FUNCTION_BLOCK fb_gm_transport
VAR_INPUT
END_VAR
VAR_OUTPUT
END_VAR
VAR
	SFCInit : bool;
	trn_lensPickUpDone: BOOL;
	trn_transportDone: BOOL;
	trn_lensSetDone: BOOL;
	var_process: INT;
	trn_homeDone: BOOL;
	trn_closeCheckDone: BOOL;
	trn_waittingLensDone: BOOL;
	retryTimer: TON;
	var_retryTimes: INT;
END_VAR

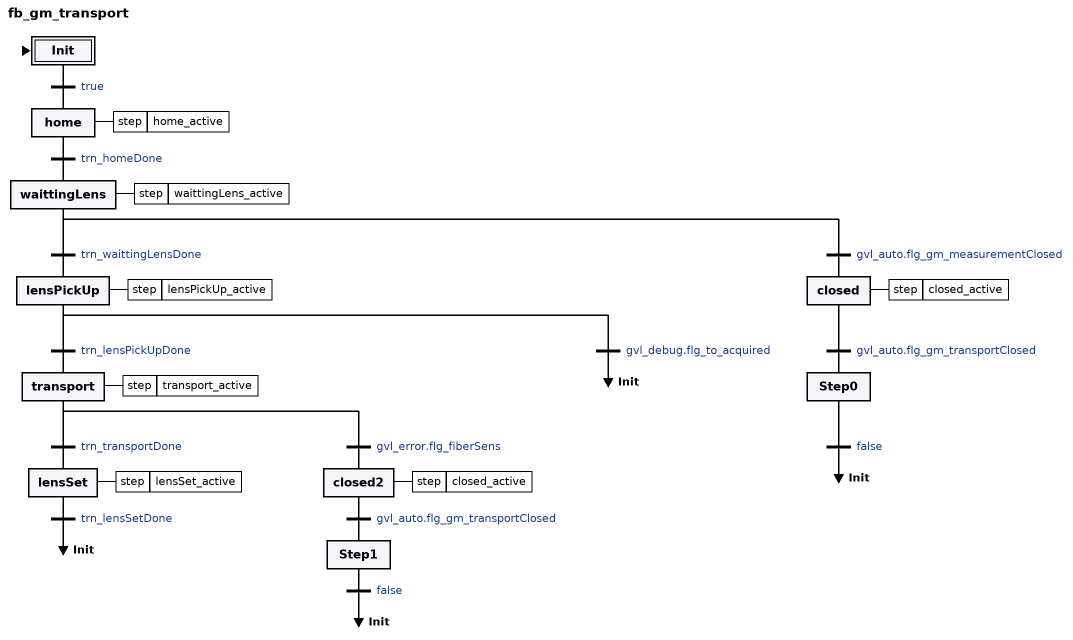
INITIAL_STEP Init:
END_STEP
TRANSITION FROM Init TO home
    := true;
END_TRANSITION
STEP home:
    home_active(N);  // step action
END_STEP
TRANSITION FROM home TO waittingLens
    := trn_homeDone;
END_TRANSITION
STEP waittingLens:
    waittingLens_active(N);  // step action
END_STEP
TRANSITION FROM waittingLens TO lensPickUp
    := trn_waittingLensDone;
END_TRANSITION
STEP lensPickUp:
    lensPickUp_active(N);  // step action
END_STEP
TRANSITION FROM lensPickUp TO transport
    := trn_lensPickUpDone;
END_TRANSITION
TRANSITION FROM lensPickUp TO Init
    := gvl_debug.flg_to_acquired;
END_TRANSITION
TRANSITION FROM waittingLens TO closed
    := gvl_auto.flg_gm_measurementClosed;
END_TRANSITION
STEP closed:
    closed_active(N);  // step action
END_STEP
TRANSITION FROM closed TO Step0
    := gvl_auto.flg_gm_transportClosed;
END_TRANSITION
STEP Step0:
END_STEP
TRANSITION FROM Step0 TO Init
    := false;
END_TRANSITION
STEP transport:
    transport_active(N);  // step action
END_STEP
TRANSITION FROM transport TO lensSet
    := trn_transportDone;
END_TRANSITION
STEP lensSet:
    lensSet_active(N);  // step action
END_STEP
TRANSITION FROM lensSet TO Init
    := trn_lensSetDone;
END_TRANSITION
TRANSITION FROM transport TO closed2
    := gvl_error.flg_fiberSens;
END_TRANSITION
STEP closed2:
    closed_active(N);  // step action
END_STEP
TRANSITION FROM closed2 TO Step1
    := gvl_auto.flg_gm_transportClosed;
END_TRANSITION
STEP Step1:
END_STEP
TRANSITION FROM Step1 TO Init
    := false;
END_TRANSITION

ACTION closed_active:
IF closed._x AND closed.x = FALSE THEN
	gvl_auto.flg_gm_transportClosed := FALSE;
ELSIF closed._x AND closed.x THEN
	gvl_auto.flg_gm_transportClosed := TRUE;
END_IF
END_ACTION

ACTION home_active:
IF home._x AND home.x = FALSE THEN
	var_process := 0;
	trn_homeDone := FALSE;
	gvl_debug.flg_to_demand:= FALSE;
ELSIF home._x AND home.x THEN
	CASE var_process OF 
		0:
			gvl_elecylinder.fbi_gm_axisPickUp.in_flg_run := FALSE;
			gvl_elecylinder.fbi_gm_axisPickUp.in_var_moveMode := eP_eleMoveMode.eleA;
			gvl_elecylinder.fbi_gm_axisTransport.in_flg_run := FALSE;
			gvl_elecylinder.fbi_gm_axisTransport.in_var_moveMode := eP_eleMoveMode.eleA;
			gvl_axis.ref_r.Execute := FALSE;
			gvl_axis.ref_r.Position := gvl_param.var_productInfo[gvl_param.var_currentProductID].teachPos.gm_rotary.origin;
			var_process := 1;
		1:
			gvl_elecylinder.fbi_gm_axisPickUp.in_flg_run := TRUE;
			gvl_elecylinder.fbi_gm_axisTransport.in_flg_run := TRUE;
			var_process := 2;
		2:
			IF gvl_elecylinder.ref_gm_axisPickUp.input.in_flg_sensA AND gvl_elecylinder.ref_gm_axisTransport.input.in_flg_sensA THEN
				gvl_elecylinder.fbi_gm_axisPickUp.in_flg_run := FALSE;
				gvl_elecylinder.fbi_gm_axisTransport.in_flg_run := FALSE;
				var_process := 3;
			END_IF
		3:
			gvl_solv.fbi_gm_pickup.in_flg_run := FALSE;
			gvl_solv.fbi_gm_pickup.in_var_moveMode := eP_svMoveMode.svA;
			var_process := 4;
		4:
			gvl_solv.fbi_gm_pickup.in_flg_run := TRUE;
			IF gvl_solv.ref_gm_pickUp.in.in_flg_sensA  THEN
				var_process := 5;
			END_IF
		5:
			gvl_auto.flg_gm_eleIsDown := FALSE;
			gvl_axis.ref_r.Execute := TRUE;
			IF gvl_axis.ref_r.Done THEN
				gvl_axis.ref_r.Execute := FALSE;
				var_process :=6;
			END_IF
		6:
			gvl_solv.fbi_gm_rotary.in_flg_run := FALSE;
			gvl_solv.fbi_gm_rotary.in_var_moveMode := eP_svMoveMode.svA;
			var_process := 7;
		7:
			gvl_solv.fbi_gm_rotary.in_flg_run := TRUE;
			IF gvl_solv.ref_gm_rotary.in.in_flg_sensA THEN
				var_process := 8;
			END_IF
		8:	
				trn_homeDone := TRUE;			
	END_CASE
END_IF
END_ACTION

ACTION lensPickUp_active:
IF lensPickUp._x AND lensPickUp.x = FALSE THEN
	gvl_axis.ref_r.Execute := FALSE;
	retryTimer.IN := FALSE;
	var_process := 0;
	var_retryTimes := 0;
	trn_lensPickUpDone := FALSE;
	gvl_auto.flg_gm_VacuumRetry := FALSE;
	gvl_solv.fbi_gm_ejector.in_flg_run := FALSE;
	gvl_solv.fbi_gm_pickup.in_flg_run := FALSE;
	gvl_solv.fbi_gm_rotary.in_flg_run := FALSE;
	gvl_elecylinder.fbi_gm_axisPickUp.in_flg_run := FALSE;
	gvl_axis.ref_r.Execute := FALSE;
ELSIF lensPickUp._x AND lensPickUp.x THEN
	CASE var_process OF 
		0:
			gvl_axis.ref_r.Position := gvl_param.var_productInfo[gvl_param.var_currentProductID].teachPos.gm_rotary.pickUp;
			gvl_axis.ref_r.Execute := TRUE;
			gvl_solv.fbi_gm_ejector.in_var_vacMode := eP_ejeVacMode.vacON;
			gvl_solv.fbi_gm_ejector.in_flg_run := TRUE;
			var_process := 1;
		1://axis theta move to pick up position
			gvl_solv.fbi_gm_ejector.in_flg_run := FALSE;
			IF gvl_axis.ref_r.Done THEN
				gvl_axis.ref_r.Execute := FALSE;
				var_process := 2;
			END_IF
		2:
			IF gvl_solv.ref_gm_ejctor.input.in_flg_sensVac THEN
				var_process := 3;
			END_IF
		3:
			gvl_solv.fbi_gm_chuck.in_var_moveMode := eP_svMoveMode.svA;
			gvl_solv.fbi_gm_push.in_var_moveMode := eP_svMoveMode.svA;
			gvl_solv.fbi_gm_chuck.in_flg_run := TRUE;
			gvl_solv.fbi_gm_push.in_flg_run := TRUE;
			var_process := 4;
		4:
			IF gvl_solv.ref_gm_chuck.in.in_flg_sensA AND gvl_solv.ref_gm_push.in.in_flg_sensA THEN
				gvl_solv.fbi_gm_chuck.in_flg_run := FALSE;
				gvl_solv.fbi_gm_push.in_flg_run := FALSE;
				var_process := 5;
			END_IF
		5:
			gvl_solv.fbi_gm_pickup.in_var_moveMode := eP_svMoveMode.svB;
			gvl_solv.fbi_gm_pickup.in_flg_run := TRUE;
			var_process := 6;
		6:
			IF gvl_solv.fbi_gm_pickup.out_flg_Done THEN
				gvl_solv.fbi_gm_pickup.in_flg_run := FALSE;
				var_process := 7;
			END_IF
		7:
			gvl_axis.ref_r.Position := gvl_param.var_productInfo[gvl_param.var_currentProductID].teachPos.gm_rotary.set;
			gvl_axis.ref_r.Execute := TRUE;
			var_process := 8;
		8:
			IF gvl_axis.ref_r.Done THEN
				gvl_axis.ref_r.Execute := FALSE;
				var_process := 9;	
			END_IF
		9:
			gvl_solv.fbi_gm_pickup.in_var_moveMode := eP_svMoveMode.svA;
			gvl_solv.fbi_gm_pickup.in_flg_run := TRUE;
			var_process := 10;
		10:
			IF gvl_solv.fbi_gm_pickup.out_flg_Done THEN
				gvl_solv.fbi_gm_pickup.in_flg_run := FALSE;
				var_process := 11;
			END_IF
		11:
			gvl_solv.fbi_gm_rotary.in_flg_run := FALSE;
			gvl_solv.fbi_gm_rotary.in_var_moveMode := eP_svMoveMode.svB;
			var_process:= 12;
		12:
			gvl_solv.fbi_gm_rotary.in_flg_run := TRUE;
			var_process := 13;
		13:
			IF gvl_solv.fbi_gm_rotary.out_flg_Done THEN
				gvl_solv.fbi_gm_rotary.in_flg_run := FALSE;
				var_process := 14;
			END_IF
		14:
			gvl_solv.fbi_gm_pickup.in_var_moveMode := eP_svMoveMode.svB;
			gvl_solv.fbi_gm_pickup.in_flg_run := TRUE;
			var_process := 15;
		15:
			IF gvl_solv.fbi_gm_pickup.out_flg_Done THEN
				gvl_solv.fbi_gm_pickup.in_flg_run := FALSE;
				var_process := 16;
			END_IF
		16:
			gvl_gm.flg_lensPickUpDone := TRUE;
			gvl_gm.var_buf_tranportCav := gvl_gm.var_buf_measurementCav;
			gvl_gm.flg_buf_gateLengthIsPassed := gvl_gm.flg_gateLengthIsPassed;
			var_process := 17;
		17:
			IF gvl_gm.flg_lensRequest AND NOT gvl_auto.flg_axisIsPcikingUp THEN
				IF gvl_debug.flg_check_quality AND gvl_debug.flg_to_stocker THEN
					gvl_debug.flg_to_demand:= TRUE;
				ELSE
					trn_lensPickUpDone := TRUE;		
				END_IF
			END_IF		
	END_CASE
END_IF
END_ACTION

ACTION lensSet_active:
IF lensSet._x AND lensSet.x = FALSE THEN
	trn_lensSetDone := FALSE;
	var_process := 0;
ELSIF lensSet._x AND lensSet.x THEN
	CASE var_process OF
		0:
			gvl_solv.fbi_gm_ejector.in_var_vacMode := eP_ejeVacMode.break;
			gvl_solv.fbi_gm_ejector.in_flg_run := FALSE;
			gvl_elecylinder.fbi_gm_axisPickUp.in_var_moveMode := eP_eleMoveMode.eleA;
			gvl_elecylinder.fbi_gm_axisPickUp.in_flg_run := FALSE;
			var_process := 1;
		1:
			gvl_solv.fbi_gm_ejector.in_flg_run := TRUE;
			IF gvl_solv.fbi_gm_ejector.out_flg_Done THEN
				gvl_solv.fbi_gm_ejector.in_flg_run := FALSE;
				var_process := 2;
			END_IF
		2:
			gvl_elecylinder.fbi_gm_axisPickUp.in_flg_run := TRUE;
			IF gvl_elecylinder.fbi_gm_axisPickUp.out_flg_Done THEN
				gvl_elecylinder.fbi_gm_axisPickUp.in_flg_run := FALSE;
				var_process := 3;
			END_IF
		3:
			gvl_gm.flg_lensSetDoneFromGM := TRUE;
			trn_lensSetDone := TRUE;
	END_CASE
END_IF
END_ACTION

PROPERTY p_Init : bool
GET
p_init := THIS^.SFCInit;
END_GET
SET
THIS^.SFCInit := p_init;
END_SET
END_PROPERTY

ACTION transport_active:
IF transport._x AND transport.x = FALSE THEN
	var_process := 0;
	trn_transportDone := FALSE;
	gvl_elecylinder.fbi_gm_axisTransport.in_flg_run := FALSE;
	gvl_elecylinder.fbi_gm_axisTransport.in_var_moveMode := eP_eleMoveMode.eleB;
	gvl_elecylinder.fbi_gm_axisPickUp.in_flg_run := FALSE;
	gvl_elecylinder.fbi_gm_axisPickUp.in_var_moveMode := eP_eleMoveMode.eleB;
	gvl_solv.fbi_gm_pickup.in_flg_run := FALSE;
	gvl_solv.fbi_gm_pickup.in_var_moveMode := eP_svMoveMode.svB;
	gvl_solv.fbi_gm_rotary.in_flg_run := FALSE;
	//gvl_solv.fbi_gm_rotary.in_var_moveMode := eP_svMoveMode.svB;
ELSIF transport._x AND transport.x THEN
	CASE var_process OF
		0:
			IF NOT gvl_auto.flg_axisIsPcikingUp THEN
				//var_process := 1;
				var_process := 3;
			END_IF
		//1:
			//gvl_solv.fbi_gm_rotary.in_flg_run := TRUE;
			//var_process := 2;
		//2:
			//IF gvl_solv.fbi_gm_rotary.out_flg_Done THEN
				//gvl_solv.fbi_gm_rotary.in_flg_run := FALSE;
				//var_process := 3;
			//END_IF
		3:
			IF NOT gvl_io.flg_fiberSens THEN
				gvl_auto.flg_gm_eleIsDown := TRUE;
				gvl_elecylinder.fbi_gm_axisTransport.in_flg_run := TRUE;
				gvl_elecylinder.fbi_gm_axisPickUp.in_flg_run := TRUE;
				gvl_solv.fbi_gm_pickup.in_flg_run := TRUE;
				var_process := 4;
			ELSE
				gvl_error.flg_fiberSens:= TRUE;
			END_IF
		4:
			IF gvl_elecylinder.fbi_gm_axisTransport.out_flg_Done THEN
				var_process := 5;
			END_IF
		5:
			gvl_elecylinder.fbi_gm_axisTransport.in_flg_run := FALSE;
			gvl_elecylinder.fbi_gm_axisPickUp.in_flg_run := FALSE;
			gvl_solv.fbi_gm_pickup.in_flg_run := FALSE;
			gvl_solv.fbi_gm_rotary.in_flg_run := FALSE;
			var_process := 6;
		6:
			trn_transportDone := TRUE;
		    
	END_CASE
END_IF
END_ACTION

ACTION waittingLens_active:
IF waittingLens._x AND waittingLens.x = FALSE THEN
	trn_waittingLensDone := FALSE;
ELSIF waittingLens._x AND waittingLens.x THEN
	IF gvl_gm.flg_requestPickup THEN
		trn_waittingLensDone := TRUE;
	END_IF
END_IF
END_ACTION

END_FUNCTION_BLOCK

(* stored: Version 1.1.0.1, ProductVersion 3.1.4024.11
   POU fb_gm_transport: Id {6860143f-ae49-4316-94c5-4ab9327b63bc}, SpecialFunc None
   Action closed_active: Id {96c65c66-3a15-482c-840c-36be55522d07}
   Action home_active: Id {88bdaa60-9fe4-442d-887d-5c200a3446ff}
   Action lensPickUp_active: Id {ceed8694-1458-4e2e-b916-92915b17d136}
   Action lensSet_active: Id {acd70e51-6aba-4b24-bf02-2aa9d180be69}
   Property p_Init: Id {10bf5141-40b0-4433-a575-d9af45a3e0b7}
   Get Get: Id {3118bc38-dfff-412b-b364-eab09bb50249}
   Set Set: Id {30a8c0fb-1e73-4e6f-ab7c-e324df64ad10}
   Action transport_active: Id {3892d2cc-fe6b-445f-90b4-be5d225098cb}
   Action waittingLens_active: Id {1be048b6-b09f-4a70-b73e-336590387d14} *)
